FUNCTION f_GetBools : LWORD
VAR_INPUT
  pArr    : POINTER TO BYTE;
  nLow    : DINT;
  nUp     : DINT;
END_VAR
VAR
  _idx    : DINT;
  _pData  : POINTER TO BYTE;
  _wRet   : LWORD;
END_VAR

FOR _idx := 0 TO nUp-1
DO
  _pData := pArr;
  IF NOT(_idx < nLow-1)
  THEN
    IF (_pData^ = 1)
    THEN
      _wRet := f_Setbit64(_wRet, _idx);
    END_IF
  END_IF
  pArr := pArr + 1;
END_FOR
f_GetBools := _wRet;

END_FUNCTION

(* stored: Version 1.1.0.1, ProductVersion 3.1.4024.9
   POU f_GetBools: Id {6edd3caa-22dd-0972-3f0b-353f2b2b83d3}, SpecialFunc None *)
